TYPE ST_ParamRecipe :
STRUCT
	stPalette1 : ST_Palette;
END_STRUCT
END_TYPE

(* stored: Version 1.1.0.1, ProductVersion 3.1.4020.12
   DUT ST_ParamRecipe: Id {d7b97810-f7a3-4f07-8edf-3767a14d55f3} *)
